# EPICS substitutions: modules/event/evrSupport/Db/ioc/IOC-IN20-IM01evr.substitutions
#==============================================================================
#
# Abs:  LCLS EVR IOC records for IN20 IM01
#
# Name: IOC-IN20-IM01evr.substitutions
#
#==============================================================================
#
file evrIMXX.db
{
pattern { DEVICE        }
	{ EVR:IN20:IM01 }
}
